FUNCTION_BLOCK E_TABLE (* Generation of a finite train of events,table driven *)
  (* Standard: 61499-1-A.11; Classification: Event Processing; Description: Generation of a finite train of events (table driven) *)
  (* Version 0.2, 2002-01-30, JHC, Rockwell Automation, SIFB version *)
  (* Version 0.1, 2001-04-29, JHC, Rockwell Automation, XML version *)
  (* Version 0.0, 1998-04-10, JHC, Rockwell Automation, SRC version *)
  (* Compiler header: package fb.rt.events; *)
  (* Compiler Java IBM VisualAge 3.0 *)
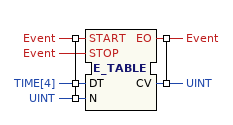
  EVENT_INPUT
    START WITH DT, N;
    STOP; (* Cancel *)
  END_EVENT
  EVENT_OUTPUT
    EO WITH CV; (* N events at periods DT,starting at DT[0]after START *)
  END_EVENT
  VAR_INPUT
    DT : ARRAY [0..3] OF TIME; (* Periods between events *)
    N : UINT; (* Number of events to generate *)
  END_VAR
  VAR_OUTPUT
    CV : UINT; (* Current event index,1 to N *)
  END_VAR
  SERVICE E_TABLE/resource
    SEQUENCE normal_operation (* N=3 *)
      E_TABLE.START(DT);
      -> E_TABLE.EO(CV=0,DT[0]after START);
      -> E_TABLE.EO(CV=1,DT[1]after previous EO);
      -> E_TABLE.EO(CV=2,DT[2]after previous EO);
    END_SEQUENCE
    SEQUENCE no_restart (* N=3 *)
      E_TABLE.START(DT);
      -> E_TABLE.EO(CV=0,DT[0]after START);
      E_TABLE.START(DT);
      -> E_TABLE.EO(CV=1,DT[1]after previous EO);
      -> E_TABLE.EO(CV=2,DT[2]after previous EO);
    END_SEQUENCE
    SEQUENCE cycle_canceled
      E_TABLE.START(DT);
      -> E_TABLE.EO(CV=0,DT[0]after START);
      E_TABLE.STOP();
    END_SEQUENCE
  END_SERVICE
END_FUNCTION_BLOCK
